FUNCTION_BLOCK BasicSKILL (* Composite Function Block Type *)
  (* Standard: 61499-2 *)
  (* Version 0.0, 1/31/2024, midxav, template *)
  PACKAGE Main;
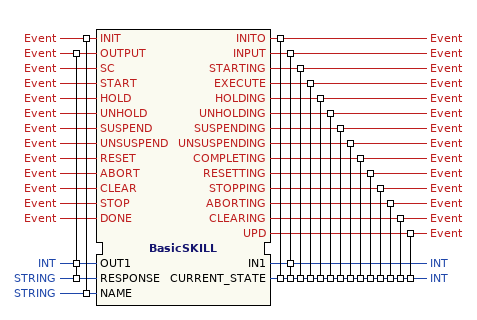
  EVENT_INPUT
    INIT WITH NAME;
    OUTPUT WITH OUT1, RESPONSE;
    SC;
    START;
    HOLD;
    UNHOLD;
    SUSPEND;
    UNSUSPEND;
    RESET;
    ABORT;
    CLEAR;
    STOP;
    DONE;
  END_EVENT
  EVENT_OUTPUT
    INITO WITH CURRENT_STATE;
    INPUT WITH IN1, CURRENT_STATE;
    STARTING WITH CURRENT_STATE;
    EXECUTE WITH CURRENT_STATE;
    HOLDING WITH CURRENT_STATE;
    UNHOLDING WITH CURRENT_STATE;
    SUSPENDING WITH CURRENT_STATE;
    UNSUSPENDING WITH CURRENT_STATE;
    COMPLETING WITH CURRENT_STATE;
    RESETTING WITH CURRENT_STATE;
    STOPPING WITH CURRENT_STATE;
    ABORTING WITH CURRENT_STATE;
    CLEARING WITH CURRENT_STATE;
    UPD WITH CURRENT_STATE;
  END_EVENT
  VAR_INPUT
    OUT1 : INT;
    RESPONSE : STRING;
    NAME : STRING;
  END_VAR
  VAR_OUTPUT
    IN1 : INT;
    CURRENT_STATE : INT;
  END_VAR
  FBS
    IThis : BasicSKILL_HMI(QI := TRUE);
    SKILL_ECC : SKILL_BFB;
  END_FBS
  EVENT_CONNECTIONS
    SKILL_ECC.STARTING TO STARTING;
    SKILL_ECC.EXECUTE TO EXECUTE;
    SKILL_ECC.HOLDING TO HOLDING;
    SKILL_ECC.UNHOLDING TO UNHOLDING;
    SKILL_ECC.SUSPENDING TO SUSPENDING;
    SKILL_ECC.UNSUSPENDING TO UNSUSPENDING;
    SKILL_ECC.COMPLETING TO COMPLETING;
    SKILL_ECC.RESETTING TO RESETTING;
    SKILL_ECC.STOPPING TO STOPPING;
    SKILL_ECC.ABORTING TO ABORTING;
    SKILL_ECC.CLEARING TO CLEARING;
    START TO SKILL_ECC.START;
    HOLD TO SKILL_ECC.HOLD;
    UNHOLD TO SKILL_ECC.UNHOLD;
    SUSPEND TO SKILL_ECC.SUSPEND;
    UNSUSPEND TO SKILL_ECC.UNSUSPEND;
    RESET TO SKILL_ECC.RESET;
    ABORT TO SKILL_ECC.ABORT;
    CLEAR TO SKILL_ECC.CLEAR;
    STOP TO SKILL_ECC.STOP;
    SC TO SKILL_ECC.SC;
    INIT TO IThis.INIT;
    OUTPUT TO IThis.OUTPUT;
    SKILL_ECC.CNF TO IThis.SKILL_OUTPUT;
    IThis.INITO TO INITO;
    IThis.INPUT TO INPUT;
    IThis.SKILL_INPUT TO SKILL_ECC.REQ;
    IThis.INITO TO IThis.SKILL_OUTPUT;
    SKILL_ECC.CNF TO UPD;
    DONE TO SKILL_ECC.DONE;
  END_CONNECTIONS
  DATA_CONNECTIONS
    OUT1 TO IThis.OUT1;
    RESPONSE TO IThis.RESPONSE;
    SKILL_ECC.CURRENT_STATE TO IThis.CURRENT_STATE;
    IThis.IN1 TO IN1;
    IThis.SKILL_CMD TO SKILL_ECC.SKILL_CMD;
    NAME TO IThis.NAME;
    SKILL_ECC.CURRENT_STATE TO CURRENT_STATE;
  END_CONNECTIONS
END_FUNCTION_BLOCK
